{attribute 'OPC.UA.DA.StructuredType' := '1'}
FUNCTION_BLOCK FB_BaseDevice

VAR
	{attribute 'OPC.UA.DA' := '1'} 
	sID: STRING; // as per P&IDs
	{attribute 'OPC.UA.DA' := '1'} 
	sDescr: STRING;
	{attribute 'OPC.UA.DA' := '1'} 
	sVarID: STRING;
	{attribute 'OPC.UA.DA' := '0'} 
	bBusy: BOOL := FALSE;
	{attribute 'OPC.UA.DA' := '1'} 
	bError: BOOL := FALSE;
	bEnable: BOOL := TRUE;
	{attribute 'OPC.UA.DA' := '1'} 
	eMode: E_DeviceMode := E_DeviceMode.AUTO;
	{attribute 'OPC.UA.DA' := '1'} 
	eState: E_DeviceState := E_DeviceState.IDLE;
	{attribute 'OPC.UA.DA' := '1'} 
	eStateTarget: E_DeviceState := E_DeviceState.IDLE;
	
	{attribute 'OPC.UA.DA' := '0'} 
	fbTONstartTime: TON;
	{attribute 'OPC.UA.DA' := '0'} 
	fbTONstopTime: TON;
	{attribute 'OPC.UA.DA' := '0'} 
	tMaxStartTime: TIME := T#5S;
	{attribute 'OPC.UA.DA' := '0'} 
	tMaxStopTime: TIME := T#5S;
	
	
	
	{attribute 'OPC.UA.DA' := '1'} 
	aErrors: ARRAY[1..10] OF ST_Alarm;	// raiseEvent() method updates Error1 / aErrors[1] only at the moment, must implement a ring buffer with error active checking for full functionality
	

END_VAR

// This is the base class for all devices (actuators and sensors)
// Provides common variables to all instances 
// Note that the I_Device interface provides the common methods for all devices

METHOD disable : BOOL
VAR_INPUT
END_VAR
bEnable := FALSE;
END_METHOD

METHOD enable : BOOL
VAR_INPUT
END_VAR
bEnable := TRUE;
END_METHOD

METHOD getCommand : E_DeviceState
VAR
	
END_VAR
getCommand := eStateTarget;
END_METHOD

METHOD getDescription : STRING
VAR_INPUT
END_VAR
getDescription := sDescr;
END_METHOD

METHOD getID : STRING
VAR_INPUT
END_VAR
getID := sID;
END_METHOD

METHOD getMode : E_DeviceMode
VAR_INPUT
END_VAR
END_METHOD

METHOD getState : E_DeviceState
VAR
	
END_VAR
getState := eState;
END_METHOD

METHOD getVarID : STRING
VAR_INPUT
END_VAR
getVarID := sVarID;
END_METHOD

METHOD inManual : BOOL
VAR_INPUT
END_VAR
IF eMode = E_DeviceMode.MANUAL THEN
	inManual := TRUE;
ELSE
	inManual := FALSE;
END_IF
END_METHOD

METHOD isEnabled : BOOL
VAR_INPUT
END_VAR
IF bEnable = TRUE THEN
	isEnabled := TRUE;
ELSE
	isEnabled := FALSE;
END_IF
END_METHOD

METHOD raiseAlarm : POINTER TO ST_Alarm
VAR_INPUT
	Priority: E_AlarmPriority; 
	Label: STRING(255);
	Enabled: BOOL := FALSE;
	DeviceAlarmID: INT; // from 1 to 10
END_VAR
aErrors[DeviceAlarmID].bEnabled := TRUE;
aErrors[DeviceAlarmID].ePriority := Priority;
aErrors[DeviceAlarmID].sLabel := Label;
END_METHOD

METHOD runSimulation : BOOL
VAR_INPUT
END_VAR
eState := eStateTarget;
END_METHOD

METHOD setCommand : BOOL
VAR_INPUT
	StateTarget: E_DeviceState;
END_VAR
eStateTarget := StateTarget;
END_METHOD

METHOD setID : BOOL
VAR_INPUT
	ID: STRING;
END_VAR
sID := ID;
END_METHOD

METHOD setMode : BOOL
VAR_INPUT
	Mode: E_DeviceMode;
END_VAR

eMode := Mode;
END_METHOD

METHOD setVarID : BOOL
VAR_INPUT
	VarID: STRING;
END_VAR
sVarID := VarID;
END_METHOD

END_FUNCTION_BLOCK

(* stored: Version 1.1.0.1, ProductVersion 3.1.4024.12
   POU FB_BaseDevice: Id {828692ff-2d6e-4df3-89c5-ba3b5a7c076d}, SpecialFunc None
   Method disable: Id {8dc51106-416a-411a-abe7-5933e106639b}
   Method enable: Id {fcf77402-d69c-4488-a625-0cd278dc8441}
   Method getCommand: Id {920e52e3-1202-46c5-a1c3-29e09b900eeb}
   Method getDescription: Id {2bc7f28a-2e61-45e7-bb68-995101606cf0}
   Method getID: Id {b64b9aca-ecb1-4a07-997e-f0ba8a4ea0e9}
   Method getMode: Id {8867d135-ce61-4e0a-ae23-dc2884cb083e}
   Method getState: Id {69dd0898-ee7b-481f-a8d8-8ec9c6401a9b}
   Method getVarID: Id {8497824c-f8dd-4aaf-b44c-cc8085f70182}
   Method inManual: Id {27c96841-69c7-4008-8e78-8fd85be25f33}
   Method isEnabled: Id {4256b052-3861-45c1-b91b-8bf8a6fd6216}
   Method raiseAlarm: Id {b7a7b830-55b5-4494-901e-92a142632bc8}
   Method runSimulation: Id {bd4de552-44f1-4903-8e42-47eb9d2b2af3}
   Method setCommand: Id {0accf221-0fb0-46a4-96c6-e8053fbf478d}
   Method setID: Id {67563d9f-305a-465c-9c60-8fd98e275a28}
   Method setMode: Id {f27b77c6-0822-44de-ae6b-8acd5d43f693}
   Method setVarID: Id {07fa29d5-9a78-4f2c-82a2-e73442a7c4ca} *)
